Universal Robots PolyScope program: move_path_3left.urp

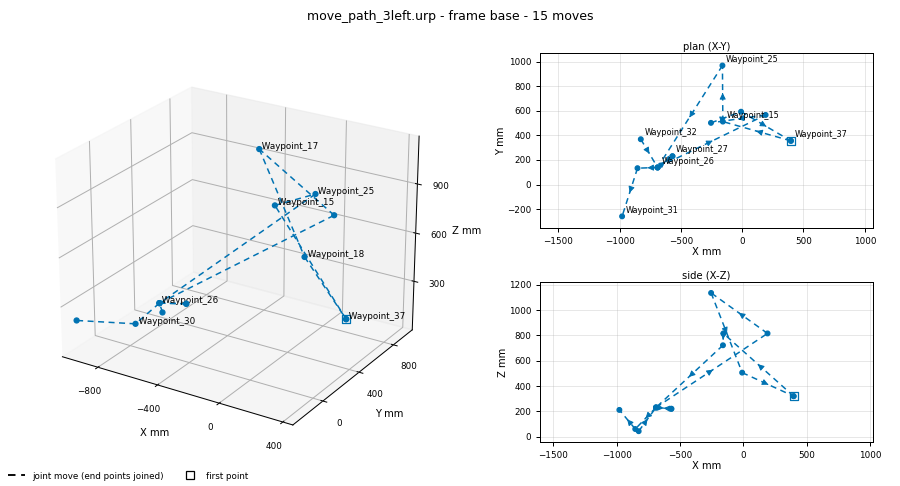
[picture p0: tool path of move_path_3left.urp in frame base, 15 of 31 moves have a stored position in this frame; points joined in program order, loops and branches not executed]
Program move_path_3left_1 (installation=default directory=/programs createdIn=5.14.5 lastSavedIn=5.14.5 robotSerialNumber=20236801216)
Calibrated DH parameters: a=[-0.000021, -0.748897, -0.28186, -0.00004, -0.000055, 0]; d=[0.236225, -424.082933, -1564.66872, 1988.95162, 0.159094, 0.153873]; alpha=[1.570844, 0.001002, 0.000337, 1.571488, -1.569996, 0]; deltaTheta=[0, -0.516316, 5.626292, 1.173211, 0.000001, 0]
InitVariablesNode variables(variable(name=freedrive_m_var, expression=False), variable(name=thread2trigger, expression=False))
Robot Program (runOnlyOnce=false)
  'this is the path for Down, Over, then Back Around'
  ''
  SafeHome (positionOptionType=SPEED_AND_ACCELERATION speed=1.047198 acceleration=1.396263 nextMotionTime=2)
  MoveJ speed 60 deg/s, acceleration 80 deg/s^2 (useActiveTCP=true) feature=Base
    Waypoint Waypoint_37: TCP in base x=397.367 y=356.259 z=319.814 mm, rx=2.3163 ry=2.0576 rz=0.0741 rad; joints [-198.126, -117.852, 133.304, -13.009, -11.423, -6.036] deg; TCP offset x=-5.49 y=-328 z=106.39 mm, rx=1.2092 ry=-1.2092 rz=1.2092 rad
    'above point is home'
    Waypoint Waypoint_15: TCP in base x=-157.621 y=513.354 z=815.678 mm, rx=-0.6727 ry=-1.8523 rz=-0.0554 rad; joints [-158.735, -104.322, 132.157, 58.275, -61.692, -46.244] deg; TCP offset x=-5.053 y=-331.71 z=103.574 mm, rx=1.2092 ry=-1.2092 rz=1.2092 rad
    Waypoint Waypoint_25: TCP in base x=-161.037 y=970.524 z=722.042 mm, rx=-0.555 ry=0.1065 rz=0.3286 rad; joints [-74.895, -76.586, 126.53, 213.07, -169.134, 52.325] deg; TCP offset x=-4.211 y=-279.829 z=105.916 mm, rx=1.2092 ry=-1.2092 rz=1.2092 rad
    Waypoint Waypoint_26: TCP in base x=-689.651 y=138.963 z=230.691 mm, rx=-0.852 ry=-1.646 rz=1.646 rad; joints [-53.938, -86.03, 160.535, 285.425, -269.23, 90.049] deg
    Waypoint Waypoint_27: TCP in base x=-568.725 y=230.602 z=220.208 mm, rx=-1.5191 ry=-0.5352 rz=0.574 rad; joints [-2.798, -73.075, 141.93, 288.829, -133.322, 87.786] deg; TCP offset x=8.385 y=-333.249 z=78.524 mm, rx=1.2092 ry=-1.2092 rz=1.2092 rad
    SuppressedNode
      Waypoint Waypoint_1: TCP in base x=-1177.596 y=138.956 z=230.69 mm, rx=-0.852 ry=-1.646 rz=1.646 rad; joints [-20.637, -63.427, 120.718, 302.664, -235.94, 90.036] deg; TCP offset x=-4.211 y=-279.829 z=105.916 mm, rx=1.2092 ry=-1.2092 rz=1.2092 rad
    SuppressedNode
      Waypoint Waypoint_2: TCP in base x=-689.651 y=138.963 z=230.691 mm, rx=-0.852 ry=-1.646 rz=1.646 rad; joints [-53.938, -86.03, 160.535, 285.425, -269.23, 90.049] deg
    SuppressedNode
      Waypoint Waypoint_3: TCP in base x=-161.037 y=970.524 z=722.042 mm, rx=-0.555 ry=0.1065 rz=0.3286 rad; joints [-74.895, -76.586, 126.53, 213.07, -169.134, 52.325] deg
    SuppressedNode
      SafeHome (positionOptionType=SPEED_AND_ACCELERATION speed=1.047198 acceleration=1.396263 nextMotionTime=2)
  ''
  p1 := pathturn[0]
  p2 := pathturn[1]
  p4 := pathturn[2]
  p5 := pathturn[3]
  pa1 := p[p1[0]+0.05,p1[1]-0.05,p1[2],p1[3],p1[4],p1[5]]
  MoveJ speed 60 deg/s, acceleration 80 deg/s^2 (useActiveTCP=true) feature=Base
    Waypoint Variable (Variable): variable=pa1
    Waypoint Variable (Variable): variable=p1
  Wait Sleep waitTime=8
  URCap WireTank Serial (WireTank Serial, WireTank, LLC) dataModel(NODE_TITLE=Serial Bridge uR1, byte_array=true, Command=[252,82,49], OUTPUT_ENTRY=Static)
  Wait Sleep waitTime=1
  MoveL speed 10 mm/s, acceleration 100 mm/s^2 (useActiveTCP=true) feature=Base
    Waypoint Variable (Variable): variable=p2
  URCap WireTank Serial (WireTank Serial, WireTank, LLC) dataModel(NODE_TITLE=Serial Bridge uR0, byte_array=true, Command=[252,82,48], OUTPUT_ENTRY=Static)
  Wait Sleep waitTime=0.5
  MoveL speed 120 mm/s, acceleration 10 mm/s^2 (useActiveTCP=true) feature=Base
    Waypoint Variable (Variable): variable=p4
  URCap WireTank Serial (WireTank Serial, WireTank, LLC) dataModel(NODE_TITLE=Serial Bridge uR1, byte_array=true, Command=[252,82,49], OUTPUT_ENTRY=Static)
  Wait Sleep waitTime=1
  MoveL speed 10 mm/s, acceleration 100 mm/s^2 (useActiveTCP=true) feature=Base
    Waypoint Variable (Variable): variable=p5
  URCap WireTank Serial (WireTank Serial, WireTank, LLC) dataModel(NODE_TITLE=Serial Bridge uR0, Command=[252,82,48], OUTPUT_ENTRY=Static, byte_array=true)
  Wait Sleep waitTime=2
  ''
  pret1 := p[p5[0]+.1,p5[1],p5[2],p5[3],p5[4],p5[5]]
  p_1 := pathturn[4]
  p_2 := pathturn[5]
  p_3 := pathturn[6]
  p_4 := pathturn[7]
  p_5 := pathturn[8]
  p_preheat := p[p_3[0]+.01,p_3[1],p_3[2],p_3[3],p_3[4],p_3[5]]
  p_pre_ret := p[p_1[0]+.03,p_1[1]-.03,p_1[2],p_1[3],p_1[4],p_1[5]]
  p_pre_ret2 := p[p_3[0]+.1,p_3[1],p_3[2],p_3[3],p_3[4],p_3[5]]
  MoveJ speed 80 deg/s, acceleration 80 deg/s^2 (useActiveTCP=true) feature=Base
    Waypoint Variable (Variable): variable=pret1
    Waypoint Waypoint_28: TCP in base x=-568.725 y=230.602 z=220.208 mm, rx=-1.5191 ry=-0.5352 rz=0.574 rad; joints [-2.798, -73.075, 141.93, 288.829, -133.322, 87.786] deg; TCP offset x=8.385 y=-333.249 z=78.524 mm, rx=1.2092 ry=-1.2092 rz=1.2092 rad
    'now go into the ccw weld position'
    Waypoint Waypoint_29: TCP in base x=-689.651 y=138.963 z=230.691 mm, rx=-0.852 ry=-1.646 rz=1.646 rad; joints [-53.938, -86.03, 160.535, 285.425, -269.23, 90.049] deg; TCP offset x=-4.211 y=-279.829 z=105.916 mm, rx=1.2092 ry=-1.2092 rz=1.2092 rad
    ''
    Waypoint Waypoint_30: TCP in base x=-853.851 y=133.267 z=60.418 mm, rx=-0.2742 ry=-2.3597 rz=0.0468 rad; joints [-34.868, -57.997, 159.687, 213.62, -283.084, 21.643] deg; TCP offset x=8.385 y=-333.249 z=78.524 mm, rx=1.2092 ry=-1.2092 rz=1.2092 rad
    Waypoint Waypoint_31: TCP in base x=-979.398 y=-259.625 z=211.289 mm, rx=-0.673 ry=-1.4594 rz=-0.6402 rad; joints [21.182, -32.844, 122.516, 179.072, -269.511, -69.331] deg
    SuppressedNode
      Waypoint Waypoint_9: TCP in base x=-161.037 y=970.524 z=722.042 mm, rx=-0.555 ry=0.1065 rz=0.3286 rad; joints [-74.895, -76.586, 126.53, 213.07, -169.134, 52.325] deg; TCP offset x=-4.211 y=-279.829 z=105.916 mm, rx=1.2092 ry=-1.2092 rz=1.2092 rad
    SuppressedNode
      Waypoint Waypoint_22: TCP in base x=-308.534 y=606.085 z=242.393 mm, rx=1.3699 ry=1.0669 rz=-1.2572 rad; joints [-84.142, -55.374, 92.791, 53.186, 94.965, 15.074] deg
  SuppressedNode
    MoveP speed 20 mm/s, acceleration 2 mm/s^2 (blendRadius=0.001 useActiveTCP=true) feature=Base
      'below (until next comment) are points for testing out ccw circle weld'
      Waypoint Waypoint_8: TCP in base x=-1291.697 y=90.422 z=23.176 mm, rx=-0.673 ry=-1.4594 rz=-0.6402 rad; joints [-2.307, -18.609, 101.914, 185.717, -269.053, -45.852] deg; TCP offset x=8.385 y=-333.249 z=78.524 mm, rx=1.2092 ry=-1.2092 rz=1.2092 rad
      Waypoint Waypoint_10: TCP in base x=-1193.179 y=196.591 z=23.164 mm, rx=-0.673 ry=-1.4594 rz=-0.6402 rad; joints [-8.888, -18.95, 110.853, 177.226, -268.954, -39.273] deg
      Waypoint Waypoint_11: TCP in base x=-1193.173 y=196.572 z=23.158 mm, rx=0.078 ry=-1.5698 rz=0.1134 rad; joints [-28.391, -18.785, 116.78, 172.699, -268.884, 35.453] deg
      'end test points'
  MoveJ speed 60 deg/s, acceleration 80 deg/s^2 (useActiveTCP=true) feature=Base
    Waypoint Variable (Variable): variable=p_pre_ret
    Waypoint Variable (Variable): variable=p_pre_ret2
    Waypoint Variable (Variable): variable=p_preheat
  Wait Sleep waitTime=8
  MoveJ speed 60 deg/s, acceleration 80 deg/s^2 (useActiveTCP=true) feature=Base
    Waypoint Variable (Variable): variable=p_pre_ret2
    Waypoint Variable (Variable): variable=p_pre_ret
  Set NoAction tcp=backofhole
  MoveL speed 50 mm/s, acceleration 1200 mm/s^2 (useActiveTCP=true) feature=Base
    Waypoint Variable (Variable): variable=p_1
  URCap WireTank Serial (WireTank Serial, WireTank, LLC) dataModel(NODE_TITLE=Serial Bridge uR1, byte_array=true, Command=[252,82,49], OUTPUT_ENTRY=Static)
  Wait Sleep waitTime=1
  MoveL speed 10 mm/s, acceleration 1200 mm/s^2 (useActiveTCP=true) feature=Base
    Waypoint Variable (Variable): variable=p_2
  MoveP speed 0.5 mm/s, acceleration 10 mm/s^2 (blendRadius=0.001 useActiveTCP=true) feature=Base
    CircleMove (OrientationMode=FIXED)
      Waypoint Variable (Variable): variable=p_3
      Waypoint Variable (Variable): variable=p_4
  MoveL speed 12 mm/s, acceleration 1200 mm/s^2 (useActiveTCP=true) feature=Base
    Waypoint Variable (Variable): variable=p_5
  URCap WireTank Serial (WireTank Serial, WireTank, LLC) dataModel(NODE_TITLE=Serial Bridge uR0, Command=[252,82,48], byte_array=true, OUTPUT_ENTRY=Static)
  Wait Sleep waitTime=2
  SuppressedNode
    MoveL speed 250 mm/s, acceleration 1200 mm/s^2 (useActiveTCP=true) feature=Base
      Waypoint Waypoint_23: TCP in base x=-540.167 y=215.949 z=34.631 mm, rx=-1.5058 ry=1.0576 rz=1.5735 rad; joints [-26.452, -65.119, 143.749, 8.723, 85.674, 218.843] deg; TCP offset x=-4.211 y=-279.829 z=105.916 mm, rx=1.2092 ry=-1.2092 rz=1.2092 rad
  SuppressedNode
    MoveJ speed 60 deg/s, acceleration 80 deg/s^2 (useActiveTCP=true) feature=Base
      Waypoint Waypoint_24: TCP in base x=-308.526 y=606.096 z=242.373 mm, rx=-2.1337 ry=0.3494 rz=2.1309 rad; joints [-107.196, -73.784, 125.643, 43.029, 90.975, 86.468] deg
  MoveJ speed 60 deg/s, acceleration 80 deg/s^2 (useActiveTCP=true) feature=Base
    Waypoint Waypoint_32: TCP in base x=-826.866 y=369.358 z=43.114 mm, rx=0.575 ry=-1.4922 rz=0.5971 rad; joints [-59.333, -19.441, 121.825, 168.37, -269.932, 102.332] deg; TCP offset x=8.385 y=-333.249 z=78.524 mm, rx=1.2092 ry=-1.2092 rz=1.2092 rad
    Waypoint Waypoint_33: TCP in base x=-689.651 y=138.963 z=230.691 mm, rx=-0.852 ry=-1.646 rz=1.646 rad; joints [-53.938, -86.03, 160.535, 285.425, -269.23, 90.049] deg; TCP offset x=-4.211 y=-279.829 z=105.916 mm, rx=1.2092 ry=-1.2092 rz=1.2092 rad
  ''
  MoveJ speed 60 deg/s, acceleration 80 deg/s^2 (useActiveTCP=true) feature=Base
    Waypoint Waypoint_16: TCP in base x=191.113 y=567.512 z=815.514 mm, rx=-0.1358 ry=0.3961 rz=0.2088 rad; joints [-94.746, -100.957, 150.262, 188.452, -152.118, 48.82] deg; TCP offset x=-5.053 y=-331.71 z=103.574 mm, rx=1.2092 ry=-1.2092 rz=1.2092 rad
    Waypoint Waypoint_17: TCP in base x=-254.566 y=502.963 z=1135.402 mm, rx=-0.2619 ry=-0.7497 rz=1.349 rad; joints [-116.61, -108.45, 141.427, 125.702, -66.866, -29.172] deg
    Waypoint Waypoint_18: TCP in base x=-9.208 y=593.718 z=505.81 mm, rx=-1.4244 ry=-2.3441 rz=-0.5276 rad; joints [-167.145, -114.278, 136.39, 39.71, -32.494, -66.269] deg
    Waypoint Waypoint_38: TCP in base x=397.38 y=356.252 z=319.817 mm, rx=2.3163 ry=2.0576 rz=0.0741 rad; joints [-198.126, -117.852, 133.304, -13.01, -11.422, -6.036] deg; TCP offset x=-5.49 y=-328 z=106.39 mm, rx=1.2092 ry=-1.2092 rz=1.2092 rad
    'above point is home'
  ''
  ''
  ''
  ''
  ''
  ''
  SafeHome (positionOptionType=SPEED_AND_ACCELERATION speed=1.047198 acceleration=1.396263 nextMotionTime=2)
